PROGRAM COUNTER
VAR
	tSensorTrig		: F_TRIG;
END_VAR

tSensorTrig(CLK := GVL.bCoilRotate);
IF tSensorTrig.Q THEN
	GVL.uRevCount1 := GVL.uRevCount1 + 1;
END_IF

IF GVL.bResetRevCount THEN
	GVL.bResetRevCount  := FALSE;
	GVL.uRevCount1		:= 0;
END_IF

GVL.uRevCount2 := REAL_TO_DINT(DINT_TO_REAL(GVL.dCountServo2) / 9216);

END_PROGRAM

(* stored: Version 1.1.0.1, ProductVersion 3.1.4024.15
   POU COUNTER: Id {e1e64f7d-cad1-4631-962a-e1effe0044d0}, SpecialFunc None *)
